// TIA Portal V18 export
VAR_GLOBAL   // PLC tag table "21_AER-SP1"
   "iAER-SP1p" AT %I12.4 : Bool;   // 1
   "iAER-SP1" AT %I12.5 : Bool;   // 1
   "iAER-SP1a" AT %I20.0 : Bool;
   "oAER-SP1p" AT %Q9.7 : Bool;
   "oAER-SP1" AT %Q12.0 : Bool;
END_VAR
